PROGRAM MAIN
VAR
	fbLiftServo: 	FB_SEW_MovidriveB;
	fbLiftArmServo:	FB_SEW_MovidriveB;
END_VAR

devicesUpdate();

METHOD devicesUpdate : BOOL
VAR_INPUT
END_VAR
fbLiftServo();
fbLiftArmServo();
END_METHOD

END_PROGRAM

(* stored: Version 1.1.0.1, ProductVersion 3.1.4024.12
   POU MAIN: Id {9f57afae-ad28-41cd-80ff-e125142449c1}, SpecialFunc None
   Method devicesUpdate: Id {3ccdbb5b-b4c7-426e-bb3f-41280683a070} *)
